TYPE UpStrOutVac_Struct :
STRUCT

	xdoUpSVac : BOOL;
	xilkUpSVac : BOOL;

END_STRUCT
END_TYPE

(* stored: Version 1.1.0.1, ProductVersion 3.1.0.24
   DUT UpStrOutVac_Struct: Id {c8cf6a41-082c-4c76-8528-bcf4ead83c40} *)
